FUNCTION_BLOCK Machine EXTENDS Composite
VAR
	subMachine01				: SubMachine1;
	subMachine02				: SubMachine2;	
	childs						: ARRAY[1..NOOFCHILDS] OF IComposite := [subMachine01,subMachine02]; 	
END_VAR
VAR CONSTANT
	NOOFCHILDS					: INT := 2;
END_VAR

METHOD logStatus
VAR
	sMessage				: STRING;		
	i						: DINT;
END_VAR
// Local status 
SUPER^.logStatus();

// Loop through childs
FOR i := 1 TO NOOFCHILDS DO
	IF childs[i]<>0 THEN
		childs[i].logStatus();
	END_IF
END_FOR
END_METHOD

END_FUNCTION_BLOCK

(* stored: Version 1.1.0.1, ProductVersion 3.1.4024.12
   POU Machine: Id {b15700fe-9243-4029-8ad1-853afcd4bec3}, SpecialFunc None
   Method logStatus: Id {c02b7963-b1ff-4852-9fd3-59e7929bf1ed} *)
